{attribute 'qualified_only'}
{attribute 'strict'}
TYPE Selector_switch :
(
	enum_member := 0
);
END_TYPE

(* stored: Version 1.1.0.1, ProductVersion 3.1.4024.12
   DUT Selector_switch: Id {4ac13029-4599-4b52-9cba-4ffdd031aef1} *)
